// TwinCAT 3 PLC project Struckig
// Title: Struckig
// Company: Stefan Besler
// Author: Stefan Besler and contributers
// ProjectVersion: 0.15.5.0
// Description: Full port of pantor ruckig library (Community version) to IEC 61131-3 Structured Text. Online Trajectory Generation. Real-time. Time-optimal. Jerk-constrained.
// ProgramVersion: 3.1.4026.18
// project tree:
//   / Constants.TcGVL (not stored), ParameterList.TcGVL (not stored)
//   Struckig/Block/ BlockInterval.TcDUT (not stored), Block.TcDUT (not stored)
//   Struckig/BrakeProfile/ BrakeProfile.TcPOU (not stored)
//   Struckig/ Integrate.TcPOU (not stored), IOtg.TcIO (not stored), Otg1.TcPOU (not stored), Otg.TcPOU
//   Struckig/Math/ BubbleSortLreal.TcPOU (not stored), Ceil.TcPOU (not stored), Clamp.TcPOU (not stored), Fmod.TcPOU (not stored), IsNaN.TcPOU (not stored), IsInfinity.TcPOU (not stored), LrealBits.TcPOU (not stored), LrealFromBits.TcPOU (not stored), Power.TcPOU (not stored), Power2.TcPOU (not stored), Cbrt.TcPOU (not stored), Roots.TcPOU (not stored)
//   Struckig/Position/ PositionFirstOrderStep1.TcPOU (not stored), PositionFirstOrderStep2.TcPOU (not stored), PositionThirdOrderStep1.TcPOU (not stored), PositionSecondOrderStep1.TcPOU (not stored), PositionThirdOrderStep2.TcPOU (not stored), PositionSecondOrderStep2.TcPOU (not stored)
//   Struckig/Profile/ ProfileDesc.TcPOU (not stored)
//   Struckig/Profile/_DataTypes/ ProfileBound.TcDUT (not stored), ProfileDirection.TcDUT (not stored), ProfileControlSigns.TcDUT (not stored), ReachedLimits.TcDUT (not stored)
//   Struckig/Velocity/ VelocitySecondOrderStep2.TcPOU (not stored), VelocityThirdOrderStep1.TcPOU (not stored), VelocitySecondOrderStep1.TcPOU (not stored), VelocityThirdOrderStep2.TcPOU (not stored)
//   Struckig/_DataTypes/ ControlInterfaceType.TcDUT (not stored), DiscretizationType.TcDUT (not stored), SynchronizationType.TcDUT (not stored), TrajectoryErrorCode.TcDUT (not stored), TrajectoryState.TcDUT (not stored)

// ---- Struckig/Otg.TcPOU
// Struckig
// Copyright (C) 2022 Stefan Besler

// This program is free software: you can redistribute it and/or modify
// it under the terms of the GNU General Public License as published by
// the Free Software Foundation, either version 3 of the License, or
// (at your option) any later version.

// This program is distributed in the hope that it will be useful,
// but WITHOUT ANY WARRANTY; without even the implied warranty of
// MERCHANTABILITY or FITNESS FOR A PARTICULAR PURPOSE.  See the
// GNU General Public License for more details.
//
// You should have received a copy of the GNU General Public License
// along with THIS PROGRAM.  IF NOT, see <http://www.gnu.org/licenses/>.
{attribute 'conditionalshow_all_locals'}
FUNCTION_BLOCK Otg IMPLEMENTS IOtg
VAR_INPUT
  CycleTime : LREAL;
  Dofs : INT;
  Enabled : ARRAY[0..ParameterList.MaxDoFs] OF BOOL;  
  ControlInterface : ControlInterfaceType := ControlInterfaceType.Position; //< The default position interface controls the full kinematic state.
  Synchronization : SynchronizationType := SynchronizationType.TimeSync; //< Synchronization behavior of multiple DoFs
  PerDofControlInterface : ARRAY[0..ParameterList.MaxDoFs] OF ControlInterfaceType; //< Per-DoF control interface (overwrites global ControlInterface)
  PerDofSynchronization: ARRAY[0..ParameterList.MaxDoFs] OF SynchronizationType; //< Per-DoF synchronization (overwrites global Synchronization)
  Discretization : DiscretizationType; //< Whether the duration should be a discrete multiple of the control cycle (off by default)
  CurrentPosition, CurrentVelocity, CurrentAcceleration : ARRAY[0..ParameterList.MaxDoFs] OF LREAL; //< Current state
  TargetPosition, TargetVelocity, TargetAcceleration : ARRAY[0..ParameterList.MaxDoFs] OF LREAL; //< Target state
  MaxVelocity : ARRAY[0..ParameterList.MaxDoFs] OF LREAL; //< Kinematic constraints
  MaxAcceleration : ARRAY[0..ParameterList.MaxDoFs] OF LREAL; //< Kinematic constraints, defaults to Infinity (Struckig.Constants.Infinity)
  MaxJerk : ARRAY[0..ParameterList.MaxDoFs] OF LREAL; //< Kinematic constraints, defaults to Infinity (Struckig.Constants.Infinity)
  MinVelocity, MinAcceleration : ARRAY[0..ParameterList.MaxDoFs] OF LREAL; //< Optional kindematic constraints
  MinDuration : LREAL := 0; //< Optional minimum duration of a trajectory. This is only considered if the Synchronization type is not none
  EnableAutoPropagate : BOOL; //< If set to true, PassOutputToInput is automatically called internally after calling the function block's body
END_VAR
VAR_OUTPUT
  NewPosition, NewVelocity, NewAcceleration, NewJerk : ARRAY[0..ParameterList.MaxDoFs] OF LREAL;
  NewCalculation : BOOL; //< Was a new trajectory calculation performed in the last cycle?
  CurrentTime : LREAL;
END_VAR
VAR
  _duration : LREAL;
  _state : TrajectoryState;  
  _inputInitialized : BOOL := FALSE;
  _newSection : INT; //< not used in Struckig, ruckig pro feature
  _blocks : ARRAY[0..ParameterList.MaxDoFs] OF Block;  
  _profiles : ARRAY[0..ParameterList.MaxDoFs] OF ProfileDesc;
  _independentMinDurations : ARRAY[0..ParameterList.MaxDoFs] OF LREAL;
  
  _positionThirdOrderStep1 : PositionThirdOrderStep1;
  _positionThirdOrderStep2 : PositionThirdOrderStep2;
  _velocityThirdOrderStep1 : VelocityThirdOrderStep1;
  _velocityThirdOrderStep2 : VelocityThirdOrderStep2;
  
  _positionSecondOrderStep1 : PositionSecondOrderStep1;
  _positionSecondOrderStep2 : PositionSecondOrderStep2;
  _velocitySecondOrderStep1 : VelocitySecondOrderStep1;
  _velocitySecondOrderStep2 : VelocitySecondOrderStep2;
  
  _positionFirstOrderStep1 : PositionFirstOrderStep1;
  _positionFirstOrderStep2 : PositionFirstOrderStep2;  
  
  _inp_min_velocity, _inp_min_acceleration : ARRAY[0..ParameterList.MaxDoFs] OF LREAL;
  _inp_per_dof_control_interface : ARRAY[0..ParameterList.MaxDoFs] OF ControlInterfaceType; //< Per-DoF control interface
  _inp_per_dof_synchronization : ARRAY[0..ParameterList.MaxDoFs] OF SynchronizationType; //< Per-DoF synchronization
  
  _dofs, _dofsEnd : INT;
  _enabled : ARRAY[0..ParameterList.MaxDoFs] OF BOOL;  
  _controlInterface : ControlInterfaceType := ControlInterfaceType.Position; //< The default position interface controls the full kinematic state.
  _synchronization : SynchronizationType := SynchronizationType.TimeSync; //< Synchronization behavior of multiple DoFs
  _perDofControlInterface : ARRAY[0..ParameterList.MaxDoFs] OF ControlInterfaceType; //< Per-DoF control interface
  _perDofSynchronization: ARRAY[0..ParameterList.MaxDoFs] OF SynchronizationType; //< Per-DoF synchronization
  _discretization : DiscretizationType; //< Whether the duration should be a discrete multiple of the control cycle (off by default)
  _currentPosition, _currentVelocity, _currentAcceleration : ARRAY[0..ParameterList.MaxDoFs] OF LREAL; //< Current state
  _targetPosition, _targetVelocity, _targetAcceleration : ARRAY[0..ParameterList.MaxDoFs] OF LREAL; //< Target state
  _maxVelocity, _maxAcceleration, _maxJerk : ARRAY[0..ParameterList.MaxDoFs] OF LREAL; //< Kinematic constraints
  _new_phase_control : ARRAY[0..ParameterList.MaxDoFs] OF LREAL;
  _minVelocity, _minAcceleration : ARRAY[0..ParameterList.MaxDoFs] OF LREAL; //< Optional kindematic constraints
  _minDuration : LREAL := 0; //< Optional minimum duration of a trajectory. This is only considered if the Synchronization type is not none
  _dt : LREAL; //< Time step between updates (cycle time) in [s]
  _errorId : INT;
  _errorMessage : STRING(255);
END_VAR

NewCalculation := FALSE;
SetBusy(TRUE);

IF NOT _inputInitialized OR_ELSE HasChanged() 
THEN
  _dofsEnd := Dofs - 1; // for looping

  Calculate();
  IF State = TrajectoryState.Error THEN
    RETURN;
  END_IF

  // Store the desired state to check for potential changes
  _dofs := Dofs;
  _enabled := Enabled;
  _controlInterface := ControlInterface;
  _synchronization := Synchronization;
  _discretization := Discretization;
  _currentPosition := CurrentPosition;
  _currentVelocity := CurrentVelocity;
  _currentAcceleration := CurrentAcceleration;
  _targetPosition := TargetPosition;
  _targetVelocity := TargetVelocity;
  _targetAcceleration := TargetAcceleration;
  _maxVelocity := MaxVelocity;
  _maxAcceleration := MaxAcceleration;
  _maxJerk := MaxJerk;
  _minVelocity := MinVelocity;
  _minAcceleration := MinAcceleration;
  _minDuration := MinDuration;
  _perDofControlInterface := PerDofControlInterface;
  _perDofSynchronization := PerDofSynchronization;
  _dt := CycleTime;
  _inputInitialized := TRUE;
  CurrentTime := 0.0;
  NewCalculation := TRUE;  
END_IF

CurrentTime := CurrentTime + _dt;
AtTime(CurrentTime, ADR(NewPosition), ADR(NewVelocity), ADR(NewAcceleration), ADR(NewJerk), ADR(_newSection));

_currentPosition := NewPosition;
_currentVelocity := NewVelocity;
_currentAcceleration := NewAcceleration;

IF CurrentTime > _duration THEN
  _state := TrajectoryState.Idle;
END_IF

IF EnableAutoPropagate
THEN
  PassOutputToInput();
END_IF

METHOD PROTECTED AbortErrorId
VAR_INPUT
  errorId : INT;
END_VAR
VAR_IN_OUT CONSTANT  
  message : STRING;
END_VAR
_state := TrajectoryState.Error;
_errorMessage := message;
_errorId := errorId;
END_METHOD

/// Get the kinematic state at a given time
{attribute 'conditionalshow'}
METHOD AtTime
VAR_INPUT
  t : LREAL;
  new_position : POINTER TO LREAL;
  new_velocity : POINTER TO LREAL;
  new_acceleration : POINTER TO LREAL;
  new_jerk : POINTER TO LREAL;
  new_section : POINTER TO INT;
END_VAR
VAR
  dof : INT;
  p : REFERENCE TO ProfileDesc;
  t_diff : LREAL;
  index : INT;
END_VAR
IF (t >= Duration) THEN
  // Keep constant acceleration
  //new_section := 1;
  FOR dof:=0 TO _dofsEnd DO
    Integrate(t - (_profiles[dof].Brake.Duration + _profiles[dof].t_sum[6]), _profiles[dof].p[7], _profiles[dof].v[7], _profiles[dof].a[7], 0, p:=new_position[dof], v:=new_velocity[dof], a:=new_acceleration[dof]);
    new_jerk[dof] := 0;
  END_FOR
  RETURN;
END_IF

//new_section := 0;
FOR dof:=0 TO _dofsEnd DO
  p REF= _profiles[dof];

  t_diff := t;
  
  // Brake pre-trajectory
  IF (p.Brake.Duration > 0) THEN
    IF (t_diff < p.Brake.Duration) THEN
      index := SEL(t_diff < p.Brake.t[0], 1, 0);
      IF (index > 0) THEN
        t_diff := t_diff - p.Brake.t[index - 1];
      END_IF

      Integrate(t_diff, p.Brake.p[index], p.Brake.v[index], p.Brake.a[index], p.Brake.j[index], p:=new_position[dof], v:=new_velocity[dof], a:=new_acceleration[dof]);
      new_jerk[dof] := p.Brake.j[index];
      CONTINUE;
    ELSE
      t_diff := t_diff - p.Brake.Duration;
    END_IF
  END_IF
  
// Accel post-trajectory
// if (new_section == profiles.size() - 1 && p.accel.duration > 0) {
//     if (t_diff_dof > p.t_sum[6]) {
//         const size_t index = (t_diff_dof < p.accel.t[0]) ? 1 : 0;
//         if (index > 0) {
//             t_diff_dof -= p.accel.t[index - 1];
//         }

//         std::tie(new_position[dof], new_velocity[dof], new_acceleration[dof]) = integrate(t_diff_dof, p.accel.p[index], p.accel.v[index], p.accel.a[index], p.accel.j[index]);
//         continue;
//     }
// }

  // Non-time synchronization
  IF (t_diff >= p.t_sum[6]) THEN
    // Keep constant acceleration
    Integrate(t_diff - p.t_sum[6], p.p[7], p.v[7], p.a[7], 0, p:=new_position[dof], v:=new_velocity[dof], a:=new_acceleration[dof]);
    new_jerk[dof] := 0;    
    CONTINUE;
  END_IF

  FOR index:=0 TO 6 DO
    IF p.t_sum[index] > t_diff
    THEN
      EXIT;
    END_IF
	END_FOR
  
  IF (index > 0) THEN
    t_diff := t_diff - p.t_sum[index - 1];
  END_IF

  Integrate(t_diff, p.p[index], p.v[index], p.a[index], p.j[index], p:=new_position[dof], v:=new_velocity[dof], a:=new_acceleration[dof]);
  new_jerk[dof] := p.j[index];      
END_FOR
END_METHOD

/// Get the kinematic state and current section at a given time without vectors for a single DoF.
/// Using this method is only allowed for DoF = 1, for higher degrees of freedom use
/// [AtTime](xref:Struckig.Otg#AtTime). Using this method for DoF > 0 will not yield any result
{attribute 'conditionalshow'}
METHOD AtTime1
VAR_INPUT
  t : LREAL;
  new_position : REFERENCE TO LREAL;
  new_velocity : REFERENCE TO LREAL;
  new_acceleration : REFERENCE TO LREAL;
  new_jerk : REFERENCE TO LREAL;  
END_VAR
IF _dofs = 1
THEN
  AtTime(t, ADR(new_position), ADR(new_velocity), ADR(new_acceleration), ADR(new_jerk), 0);
END_IF
END_METHOD

METHOD PRIVATE Calculate
VAR_INST
  dof, i : INT;
  p, p_limiting : REFERENCE TO ProfileDesc;
  found_profile : BOOL;
  limiting_dof : INT := -1; // The DoF that doesn't need step 2
  discrete_duration, found_synchronization, found_time_synchronization : BOOL;
  t_profile : LREAL;
  noneSynchronizationCount, phaseSychronizations, phaseOrNoneSychronizationCount : INT;
  has_zero_limits : BOOL;
END_VAR
SetBusy(TRUE);
IF NOT ValidateInputOrAbort(checkCurrentStateWithinLimits:=FALSE, checkTargetStateWithinLimits:=TRUE)
THEN
  RETURN;
END_IF

FOR dof:=0 TO _dofsEnd
DO
  p REF=_profiles[dof];
  
  _inp_min_velocity[dof] := SEL(ABS(MinVelocity[dof]) < Constants.Epsilon, MinVelocity[dof], -MaxVelocity[dof]);
  _inp_min_acceleration[dof] := SEL(ABS(MinAcceleration[dof]) < Constants.Epsilon, MinAcceleration[dof], -MaxAcceleration[dof]);
  _inp_per_dof_control_interface[dof] := SEL(PerDofControlInterface[dof] = ControlInterfaceType.Undefined, PerDofControlInterface[dof], ControlInterface);
  _inp_per_dof_synchronization[dof] := SEL(PerDofSynchronization[dof] = SynchronizationType.Undefined, PerDofSynchronization[dof], Synchronization); 
  
  IF NOT Enabled[dof]
  THEN
    p.p[7] := CurrentPosition[dof];
    p.v[7] := CurrentVelocity[dof];
    p.a[7] := CurrentAcceleration[dof];    
    p.t_sum[6] := 0.0;
    _blocks[dof].Tmin := 0.0;
    _blocks[dof].A.IsUsed := FALSE;
    _blocks[dof].B.IsUsed := FALSE;    
    CONTINUE;
	END_IF
  
  CASE _inp_per_dof_control_interface[dof]
  OF
    ControlInterfaceType.Position:
    
      IF NOT IsInfinity(MaxJerk[dof])
      THEN
        p.Brake.PositionBrakeTrajectory(CurrentVelocity[dof], CurrentAcceleration[dof], MaxVelocity[dof], _inp_min_velocity[dof], MaxAcceleration[dof], _inp_min_acceleration[dof], MaxJerk[dof]);
      ELSIF NOT IsInfinity(MaxAcceleration[dof])
      THEN
        p.Brake.SecondOrderPositionBrakeTrajectory(CurrentVelocity[dof], MaxVelocity[dof], _inp_min_velocity[dof], MaxAcceleration[dof], _inp_min_acceleration[dof]);
      END_IF    

      p.SetBoundaryPosition(CurrentPosition[dof], CurrentVelocity[dof], CurrentAcceleration[dof], TargetPosition[dof], TargetVelocity[dof], TargetAcceleration[dof]);

    ControlInterfaceType.Velocity:
      IF NOT IsInfinity(MaxJerk[dof])
      THEN    
        p.Brake.VelocityBrakeTrajectory(CurrentVelocity[dof], CurrentAcceleration[dof], MaxAcceleration[dof], _inp_min_acceleration[dof], MaxJerk[dof]);
      ELSIF NOT IsInfinity(MaxAcceleration[dof])
      THEN
        p.Brake.SecondOrderVelocityBrakeTrajectory();        
      END_IF
      
      p.SetBoundaryVelocity(CurrentPosition[dof], CurrentVelocity[dof], CurrentAcceleration[dof], TargetVelocity[dof], TargetAcceleration[dof]);      
	END_CASE
  
  IF NOT IsInfinity(MaxJerk[dof])
  THEN
    p.Brake.Finalize(p.p[0], p.v[0], p.a[0]);
  ELSIF NOT IsInfinity(MaxAcceleration[dof])
  THEN
    p.Brake.FinalizeSecondOrder(p.p[0], p.v[0], p.a[0]);    
  END_IF

  CASE _inp_per_dof_control_interface[dof]
  OF
    ControlInterfaceType.Position:
      IF NOT IsInfinity(MaxJerk[dof])
      THEN
        _positionThirdOrderStep1.Set(p.p[0], p.v[0], p.a[0], p.pf, p.vf, p.af, MaxVelocity[dof], _inp_min_velocity[dof], MaxAcceleration[dof], _inp_min_acceleration[dof], MaxJerk[dof]);
        found_profile := _positionThirdOrderStep1.Get(p, _blocks[dof]);      
      ELSIF NOT IsInfinity(MaxAcceleration[dof])
      THEN
        _positionSecondOrderStep1.Set(p.p[0], p.v[0], p.pf, p.vf, MaxVelocity[dof], _inp_min_velocity[dof], MaxAcceleration[dof], _inp_min_acceleration[dof]);
        found_profile := _positionSecondOrderStep1.Get(p, _blocks[dof]);          
      ELSE
        _positionFirstOrderStep1.Set(p.p[0], p.pf, MaxVelocity[dof], _inp_min_velocity[dof]);
        found_profile := _positionFirstOrderStep1.Get(p, _blocks[dof]);          
      END_IF

    ControlInterfaceType.Velocity:
      IF NOT IsInfinity(MaxJerk[dof])
      THEN    
        _velocityThirdOrderStep1.Set(p.v[0], p.a[0], p.vf, p.af, MaxAcceleration[dof], _inp_min_acceleration[dof], MaxJerk[dof]);
        found_profile := _velocityThirdOrderStep1.Get(p, _blocks[dof]);
      ELSIF NOT IsInfinity(MaxAcceleration[dof])
      THEN
        _velocitySecondOrderStep1.Set(p.v[0], p.vf, MaxAcceleration[dof], _inp_min_acceleration[dof]);
        found_profile := _velocitySecondOrderStep1.Get(p, _blocks[dof]);    
      END_IF  
	END_CASE
  
  IF NOT found_profile
  THEN
    has_zero_limits := (MaxAcceleration[dof] = 0.0 OR_ELSE _inp_min_acceleration[dof] = 0.0 OR_ELSE MaxJerk[dof] = 0.0);
    IF has_zero_limits
    THEN
      AbortErrorId(TrajectoryErrorCode.ZeroLimitsConflict, '');
      RETURN;
    ELSE 
      AbortErrorId(TrajectoryErrorCode.CalculateStep1Failed, '');      
      RETURN;
    END_IF
	END_IF

  _independentMinDurations[dof] := _blocks[dof].Tmin;
END_FOR


discrete_duration := (Discretization = DiscretizationType.Discrete);

IF (dofs = 0 AND_THEN MinDuration <> 0 AND_THEN discrete_duration <> 0)
THEN 
  _duration := _blocks[0].Tmin;
  _profiles[0] := _blocks[0].Pmin;
  RETURN;
END_IF

found_synchronization := Synchronize(discrete_duration, MinDuration, _duration, limiting_dof);
IF NOT found_synchronization
THEN
  has_zero_limits := FALSE;
  FOR i:=0 TO _dofsEnd
  DO
    IF MaxAcceleration[dof] = 0.0 OR_ELSE _inp_min_acceleration[dof] = 0.0 OR_ELSE MaxJerk[dof] = 0.0
    THEN
      has_zero_limits := TRUE;
      EXIT;
    END_IF
  END_FOR
      
  IF has_zero_limits
  THEN
    AbortErrorId(TrajectoryErrorCode.ZeroLimitsConflictInSynchronization, '');
    RETURN;
  ELSE
    AbortErrorId(TrajectoryErrorCode.SynchronizationFailed, '');
    RETURN;    
	END_IF    
END_IF

// None Synchronization
FOR dof:=0 TO _dofsEnd
DO
  IF Enabled[dof] AND_THEN _inp_per_dof_synchronization[dof] = SynchronizationType.None
  THEN
    _profiles[dof] := _blocks[dof].Pmin;
    IF _blocks[dof].Tmin > Duration
    THEN
      _duration := _blocks[dof].Tmin;
      limiting_dof := dof;
    END_IF
  END_IF
END_FOR

IF (Duration = 0.0) THEN
  // Copy all profiles for end state
  FOR dof:=0 TO _dofsEnd
  DO
    _profiles[dof] := _blocks[dof].Pmin;
  END_FOR
  RETURN;
END_IF

noneSynchronizationCount := -1;
phaseSychronizations := -1;
phaseOrNoneSychronizationCount := -1;
FOR dof:=0 TO _dofsEnd DO 
  IF _inp_per_dof_synchronization[dof] = SynchronizationType.None
  THEN
    noneSynchronizationCount := noneSynchronizationCount + 1;
    phaseOrNoneSychronizationCount := phaseOrNoneSychronizationCount + 1;
  ELSIF _inp_per_dof_synchronization[dof] = SynchronizationType.Phase
  THEN
    phaseOrNoneSychronizationCount := phaseOrNoneSychronizationCount + 1;
    phaseSychronizations := phaseSychronizations + 1;
  END_IF
END_FOR

IF NOT discrete_duration AND_THEN noneSynchronizationCount = _dofsEnd
THEN
  RETURN;
END_IF

IF limiting_dof >= 0 AND_THEN phaseSychronizations >= 0 THEN
  p_limiting REF= _profiles[limiting_dof];
  IF IsInputCollinear(p_limiting.Direction, limiting_dof, _new_phase_control) THEN
    found_time_synchronization := TRUE;
    FOR dof:=0 TO _dofsEnd DO
      IF NOT Enabled[dof] OR_ELSE dof = limiting_dof OR_ELSE _inp_per_dof_synchronization[dof] <> SynchronizationType.Phase THEN
        CONTINUE;
      END_IF

      p REF= _profiles[dof];
      t_profile := Duration - p.Brake.Duration - p.Accel.Duration;

      p.t := p_limiting.t; // Copy timing information from limiting DoF
      p.ControlSigns := p_limiting.ControlSigns;

      CASE _inp_per_dof_control_interface[dof]
      OF
        ControlInterfaceType.Position:
          CASE p.ControlSigns
          OF
            ProfileControlSigns.Uddu:
            
              IF NOT IsInfinity(MaxJerk[dof])
              THEN
                IF NOT p.CheckWithTiming2(ProfileControlSigns.Uddu, ReachedLimits.None, t_profile, _new_phase_control[dof], MaxVelocity[dof], _inp_min_velocity[dof], MaxAcceleration[dof], _inp_min_acceleration[dof], MaxJerk[dof])
                THEN
                  found_time_synchronization := FALSE;                        
                END_IF
              ELSIF NOT IsInfinity(MaxAcceleration[dof])
              THEN
                IF NOT p.CheckForSecondOrderWithTiming2(ProfileControlSigns.Uddu, ReachedLimits.None, t_profile, _new_phase_control[dof], -_new_phase_control[dof], MaxVelocity[dof], _inp_min_velocity[dof], MaxAcceleration[dof], _inp_min_acceleration[dof])
                THEN
                  found_time_synchronization := FALSE;                        
                END_IF
              ELSE
                IF NOT p.CheckForFirstOrderWithTiming2(ProfileControlSigns.Uddu, ReachedLimits.None, t_profile, _new_phase_control[dof], MaxVelocity[dof], _inp_min_velocity[dof])
                THEN
                  found_time_synchronization := FALSE;                        
                END_IF
              END_IF
            
            ProfileControlSigns.Udud:
              IF NOT IsInfinity(MaxJerk[dof])
              THEN            
                IF NOT p.CheckWithTiming2(ProfileControlSigns.Udud, ReachedLimits.None, t_profile, _new_phase_control[dof], MaxVelocity[dof], _inp_min_velocity[dof], MaxAcceleration[dof], _inp_min_acceleration[dof], MaxJerk[dof])
                THEN            
                  found_time_synchronization := FALSE;
                END_IF
              ELSE
                IF NOT p.CheckForSecondOrderWithTiming2(ProfileControlSigns.Udud, ReachedLimits.None, t_profile, _new_phase_control[dof], -_new_phase_control[dof], MaxVelocity[dof], _inp_min_velocity[dof], MaxAcceleration[dof], _inp_min_acceleration[dof])
                THEN
                  found_time_synchronization := FALSE;                        
                END_IF
              END_IF                
          END_CASE
        
        ControlInterfaceType.Velocity:
          CASE p.ControlSigns
          OF
            ProfileControlSigns.Uddu:
            
              IF NOT IsInfinity(MaxJerk[dof])
              THEN  
                IF NOT p.CheckForVelocityWithTiming(ProfileControlSigns.Uddu, ReachedLimits.None, _new_phase_control[dof], MaxAcceleration[dof], _inp_min_acceleration[dof], MaxJerk[dof])
                THEN
                  found_time_synchronization := FALSE;                        
                END_IF
              ELSE
                IF NOT p.CheckForSecondOrderVelocityWithTiming2(ProfileControlSigns.Uddu, ReachedLimits.None, t_profile, _new_phase_control[dof], MaxAcceleration[dof], _inp_min_acceleration[dof])
                THEN
                  found_time_synchronization := FALSE;                        
                END_IF
              END_IF
          
            ProfileControlSigns.Udud:
            
              IF NOT IsInfinity(MaxJerk[dof])
              THEN             
                IF NOT p.CheckForVelocityWithTiming(ProfileControlSigns.Udud, ReachedLimits.None, _new_phase_control[dof], MaxAcceleration[dof], _inp_min_acceleration[dof], MaxJerk[dof])
                THEN            
                  found_time_synchronization := FALSE;
                END_IF
              ELSE
                IF NOT p.CheckForSecondOrderVelocityWithTiming2(ProfileControlSigns.Udud, ReachedLimits.None, t_profile, _new_phase_control[dof], MaxAcceleration[dof], _inp_min_acceleration[dof])
                THEN
                  found_time_synchronization := FALSE;                        
                END_IF
              END_IF                
          END_CASE        
      END_CASE
  

      p.Limits := p_limiting.Limits; // After check method call to set correct limits
    END_FOR

    IF found_time_synchronization AND_THEN phaseOrNoneSychronizationCount = _dofsEnd  THEN
      RETURN;
    END_IF
  END_IF
END_IF

// Time Synchronization
FOR dof:=0 TO _dofsEnd
DO
  IF NOT Enabled[dof] OR_ELSE ((dof = limiting_dof OR_ELSE _inp_per_dof_synchronization[dof] = SynchronizationType.None) AND_THEN NOT discrete_duration) THEN
    CONTINUE;
  END_IF
  
  p REF= _profiles[dof];
  t_profile := Duration - p.Brake.Duration - p.Accel.Duration;
  
  IF (_inp_per_dof_synchronization[dof] = SynchronizationType.TimeIfNecessarySync AND_THEN ABS(TargetVelocity[dof]) < Constants.Epsilon AND_THEN ABS(CurrentAcceleration[dof]) < Constants.Epsilon) THEN
      p := _blocks[dof].Pmin;
      CONTINUE;
  END_IF
  
  // Check if the final time corresponds to an extremal profile calculated in step 1
  // Use 2*eps because of numerical robustness in duration discretization
  IF (ABS(t_profile - _blocks[dof].Tmin) < Constants.Epsilon) THEN
      p := _blocks[dof].Pmin;
      CONTINUE;
  ELSIF (_blocks[dof].A.IsUsed AND_THEN ABS(t_profile - _blocks[dof].A.Right) < 2 * Constants.Epsilon16)
  THEN
      p := _blocks[dof].A.Profile;
      CONTINUE;
  ELSIF (_blocks[dof].B.IsUsed AND_THEN ABS(t_profile - _blocks[dof].B.Right) < 2 * Constants.Epsilon16)
  THEN
      p := _blocks[dof].B.Profile;
      CONTINUE;
  END_IF
  
  CASE (_inp_per_dof_control_interface[dof])
  OF  
    ControlInterfaceType.Position: 
    
      IF NOT IsInfinity(MaxJerk[dof])
      THEN       
        _positionThirdOrderStep2.Set(t_profile, p.p[0], p.v[0], p.a[0], p.pf, p.vf, p.af, MaxVelocity[dof], _inp_min_velocity[dof], MaxAcceleration[dof], _inp_min_acceleration[dof], MaxJerk[dof]);
        found_time_synchronization := _positionThirdOrderStep2.Get(p);
      ELSIF NOT IsInfinity(MaxAcceleration[dof])
      THEN
        _positionSecondOrderStep2.Set(t_profile, p.p[0], p.v[0], p.pf, p.vf, MaxVelocity[dof], _inp_min_velocity[dof], MaxAcceleration[dof], _inp_min_acceleration[dof]);
        found_time_synchronization := _positionSecondOrderStep2.Get(p);        
      ELSE
        _positionFirstOrderStep2.Set(t_profile, p.p[0], p.pf, MaxVelocity[dof], _inp_min_velocity[dof]);
        found_time_synchronization := _positionFirstOrderStep2.Get(p);        
      END_IF

    ControlInterfaceType.Velocity: 
      IF NOT IsInfinity(MaxJerk[dof])
      THEN    
        _velocityThirdOrderStep2.Set(t_profile, p.v[0], p.a[0], p.vf, p.af, MaxAcceleration[dof], _inp_min_acceleration[dof], MaxJerk[dof]);
        found_time_synchronization := _velocityThirdOrderStep2.Get(p);
      ELSE
        _velocitySecondOrderStep2.Set(t_profile, p.v[0], p.vf, MaxAcceleration[dof], _inp_min_acceleration[dof]);
        found_time_synchronization := _velocitySecondOrderStep2.Get(p);
      END_IF
  END_CASE

  IF NOT found_time_synchronization
  THEN
    AbortErrorId(TrajectoryErrorCode.SynchronizationFailed, '');
    RETURN;
  END_IF
END_FOR
END_METHOD

/// This method simply calls the body of the function block
METHOD Cyclic
VAR_INPUT
END_VAR
THIS^();
END_METHOD

PROPERTY Duration : LREAL
GET
Duration := _duration;
END_GET
END_PROPERTY

METHOD ErrorCode : TrajectoryErrorCode
VAR_INPUT
END_VAR
ErrorCode := _errorId;
END_METHOD

METHOD ErrorMessage : STRING(255)
VAR_INPUT
END_VAR
IF _errorMessage = ''
THEN
  CASE _errorId
  OF
    TrajectoryErrorCode.CalculateStep1Failed: ErrorMessage := 'Trajectory generation failed in step1';
    TrajectoryErrorCode.InvalidInput: ErrorMessage := 'Trajectory-generation invalid input';
    TrajectoryErrorCode.SynchronizationFailed: ErrorMessage := 'Trajectory-generation synchronization failed';
    TrajectoryErrorCode.ZeroLimitsConflict: ErrorMessage := 'Zero limits conflict in step 1';
    TrajectoryErrorCode.ZeroLimitsConflictInSynchronization: ErrorMessage := 'Zero limits conflict with other degrees of freedom in time synchronization';

  ELSE
    IF State = TrajectoryState.Error
    THEN
      ErrorMessage := 'Unknown error';
    END_IF
  END_CASE
ELSE
  ErrorMessage := _errorMessage;
END_IF
END_METHOD

METHOD FB_init : BOOL
VAR_INPUT
	bInitRetains : BOOL; // if TRUE, the retain variables are initialized (warm start / cold start)
	bInCopyCode : BOOL;  // if TRUE, the instance afterwards gets moved into the copy code (online change)
  cycletime : LREAL;
  dofs : SINT;
END_VAR
VAR
  i : INT;
  blockSize : UDINT := SIZEOF(Block)*SINT_TO_UDINT(dofs);
  profileSize : UDINT :=  SIZEOF(ProfileDesc)*SINT_TO_UDINT(dofs);  
END_VAR
THIS^.Dofs := dofs;

FOR i:=0 TO ParameterList.MaxDoFs
DO
  Enabled[i] := i < dofs;
  MaxAcceleration[i] := Constants.Infinity;  
  MaxJerk[i] := Constants.Infinity;
END_FOR
_dt := THIS^.CycleTime := cycletime;
END_METHOD

METHOD PRIVATE HasChanged : BOOL
VAR
  i : INT;  
END_VAR
IF _dofs <> Dofs
THEN
  HasChanged := TRUE;
  RETURN;
END_IF

FOR i:=0 TO _dofsEnd
DO
  IF NOT (_currentPosition[i] = CurrentPosition[i] AND_THEN
     _currentVelocity[i] = CurrentVelocity[i] AND_THEN
     _currentAcceleration[i] = CurrentAcceleration[i] AND_THEN
     _targetPosition[i] = TargetPosition[i] AND_THEN
     _targetVelocity[i] = TargetVelocity[i] AND_THEN
     _targetAcceleration[i] = TargetAcceleration[i] AND_THEN
     _maxVelocity[i] = MaxVelocity[i] AND_THEN
     _maxAcceleration[i] = MaxAcceleration[i] AND_THEN
     _maxJerk[i] = MaxJerk[i] AND_THEN
     _enabled[i] = Enabled[i] AND_THEN
     _minVelocity[i] = MinVelocity[i] AND_THEN
     _minAcceleration[i] = MinAcceleration[i] AND_THEN
     _perDofControlInterface[i] = PerDofControlInterface[i] AND_THEN
     _perDofSynchronization[i] = PerDofSynchronization[i])
  THEN
    HasChanged := TRUE;  
    RETURN;
	END_IF
END_FOR

IF NOT (_controlInterface = ControlInterface AND_THEN
   _synchronization = Synchronization AND_THEN
   _discretization = Discretization AND_THEN
   _minDuration = MinDuration)   
THEN
  HasChanged := TRUE;
  RETURN;
END_IF
END_METHOD

METHOD INTERNAL IsBlocked : BOOL
VAR_INPUT
  block : REFERENCE TO Block;
  t : LREAL;
END_VAR
IsBlocked := (t < block.Tmin) OR_ELSE (block.A.IsUsed AND_THEN block.A.Left < t AND_THEN t < block.A.Right) OR_ELSE (block.B.IsUsed AND_THEN block.B.Left < t AND_THEN t < block.B.Right);
END_METHOD

/// Is the trajectory (in principle) phase synchronizable?
METHOD INTERNAL IsInputCollinear : BOOL
VAR_INPUT
  limitingDirection : ProfileDirection;
  limitingDof : INT;
  new_phase_control : REFERENCE TO ARRAY[0..ParameterList.MaxDoFs] OF LREAL;
END_VAR
VAR_INST
  scale_dof : INT := -1;
  dof : INT;
  pd : ARRAY[0..ParameterList.MaxDoFs] OF LREAL;
  scale_vector : POINTER TO LREAL;
  pd_scale, v0_scale, a0_scale, vf_scale, af_scale, scale, scale_limiting, current_scale : LREAL;
  control_limiting : LREAL;
END_VAR
// Check that vectors pd, v0, a0, vf, af are collinear
FOR dof:=0 TO _dofsEnd
DO
  pd[dof] := TargetPosition[dof] - CurrentPosition[dof];
END_FOR

scale_dof := -1;
FOR dof:=0 TO _dofsEnd
DO
  IF _inp_per_dof_synchronization[dof] <> SynchronizationType.Phase
  THEN
    CONTINUE;
	END_IF
  
  IF _inp_per_dof_control_interface[dof] = ControlInterfaceType.Position AND_THEN ABS(pd[dof]) > Constants.Epsilon
  THEN
    scale_vector := ADR(pd);
    scale_dof := dof;
    EXIT;

  ELSIF ABS(CurrentVelocity[dof]) > Constants.Epsilon
  THEN
    scale_vector := ADR(CurrentVelocity);
    scale_dof := dof;
    EXIT;

  ELSIF ABS(CurrentAcceleration[dof]) >  Constants.Epsilon
  THEN
    scale_vector := ADR(CurrentAcceleration);
    scale_dof := dof;
    EXIT;
  
  ELSIF ABS(TargetVelocity[dof]) >  Constants.Epsilon
  THEN
    scale_vector := ADR(TargetVelocity);
    scale_dof := dof;
    EXIT;

  ELSIF ABS(TargetAcceleration[dof]) > Constants.Epsilon
  THEN
    scale_vector := ADR(TargetAcceleration);
    scale_dof := dof;
    EXIT;
  END_IF
END_FOR

IF scale_dof < 0
THEN
  RETURN; // Zero everywhere is in theory collinear, but that trivial case is better handled elsewhere
END_IF

scale := scale_vector[scale_dof];
pd_scale := pd[scale_dof] / scale;
v0_scale := CurrentVelocity[scale_dof] / scale;
vf_scale := TargetVelocity[scale_dof] / scale;
a0_scale := CurrentAcceleration[scale_dof] / scale;
af_scale := TargetAcceleration[scale_dof] / scale;

scale_limiting := scale_vector[limitingDof];
control_limiting := SEL(limitingDirection = ProfileDirection.Up, -MaxJerk[limitingDof], MaxJerk[limitingDof]);

IF IsInfinity(MaxJerk[limitingDof])
THEN
  control_limiting := SEL(limitingDirection = ProfileDirection.Up, _inp_min_acceleration[limitingDof], MaxAcceleration[limitingDof]);
END_IF

IF ABS(scale_limiting) < Constants.Epsilon
THEN
  RETURN;
END_IF

FOR dof:=0 TO _dofsEnd
DO
  IF _inp_per_dof_synchronization[dof] <> SynchronizationType.Phase
  THEN
    CONTINUE;
	END_IF
  
  current_scale := scale_vector[dof];
  IF (_inp_per_dof_control_interface[dof] = ControlInterfaceType.Position AND_THEN ABS(pd[dof] - pd_scale * current_scale) > Constants.Epsilon)
    OR_ELSE ABS(CurrentVelocity[dof] - v0_scale * current_scale) > Constants.Epsilon
    OR_ELSE ABS(CurrentAcceleration[dof] - a0_scale * current_scale) > Constants.Epsilon
    OR_ELSE ABS(TargetVelocity[dof] - vf_scale * current_scale) > Constants.Epsilon
    OR_ELSE ABS(TargetAcceleration[dof] - af_scale * current_scale) > Constants.Epsilon
  THEN
    RETURN;
	END_IF
  
  new_phase_control[dof] := control_limiting * current_scale / scale_limiting;
END_FOR

IsInputCollinear := TRUE;
END_METHOD

METHOD PassOutputToInput
VAR_INPUT
END_VAR
CurrentPosition := NewPosition;
CurrentVelocity := NewVelocity;
CurrentAcceleration := NewAcceleration;

// Remove first intermediate waypoint if section did change
// not supported in Struckig, this is a Ruckig Pro Feature
//IF HasSectionChanged AND_THEN IntermediatePositionCount > 0
//THEN
//  IntermediatePositionIndex := IntermediatePositionIndex + 1;
//END_IF
END_METHOD

/// Resets the instance (e.g. to force a new calculation on the next update).
/// This method can be used to trigger a new trajectory even if inputs do not change.
METHOD Reset
VAR_INPUT
END_VAR
_inputInitialized := FALSE;
END_METHOD

METHOD PROTECTED SetBusy
VAR_INPUT
  on : BOOL;
END_VAR
_state := TrajectoryState.Busy;
END_METHOD

PROPERTY State : TrajectoryState
GET
State := _state;
END_GET
END_PROPERTY

METHOD INTERNAL Synchronize : BOOL
VAR_INPUT
  discrete_duration : BOOL;
END_VAR
VAR_IN_OUT
  Tmin : LREAL;
  t_sync : LREAL;
  limiting_dof : INT;
END_VAR
VAR_INST
  possible_t_syncs : ARRAY [0..3*ParameterList.MaxDoFs] OF LREAL;
  idx : ARRAY [0..3*ParameterList.MaxDoFs] OF INT;  
  idx_end : INT;
  possible_t_sync : REFERENCE TO LREAL;
  any_interval : BOOL;
  dof : INT;
  i,j, h : INT;
  is_blocked : BOOL;
  remainder : LREAL;
END_VAR
// Possible t_syncs are the start times of the intervals and optional Tmin
any_interval := FALSE;
FOR dof := 0 TO _dofsEnd
DO
  // Ignore DoFs without synchronization here
  IF _inp_per_dof_synchronization[dof] = SynchronizationType.None
  THEN
    possible_t_syncs[dof] := 0;
    possible_t_syncs[Dofs + dof] := Constants.Infinity;
    possible_t_syncs[2 * Dofs + dof] := Constants.Infinity;
  ELSE
    possible_t_syncs[dof] := _blocks[dof].Tmin;
    possible_t_syncs[Dofs + dof] := SEL(_blocks[dof].A.IsUsed, Constants.Infinity, _blocks[dof].A.Right);
    possible_t_syncs[2 * Dofs + dof] := SEL(_blocks[dof].B.IsUsed, Constants.Infinity, _blocks[dof].B.Right);
    any_interval := any_interval OR_ELSE _blocks[dof].A.IsUsed OR_ELSE _blocks[dof].B.IsUsed;
  END_IF
END_FOR

possible_t_syncs[3 * Dofs] := SEL(Tmin = 0, Tmin, Constants.Infinity);
any_interval := any_interval OR_ELSE Tmin > 0;
IF discrete_duration
THEN
  FOR i:=0 TO 3*Dofs-1
  DO
    possible_t_sync REF= possible_t_syncs[i];
    IF possible_t_sync = Constants.Infinity
    THEN
      CONTINUE;
		END_IF
    
    remainder := Fmod(possible_t_sync, CycleTime); // in [0, delta_time)
    IF remainder > Constants.Epsilon16 THEN
      possible_t_sync := possible_t_sync + CycleTime - remainder;
    END_IF     
  END_FOR
END_IF

// Bubblesort possible_t_syncs from best to worst
idx_end := SEL(any_interval, _dofsEnd, 3*DOFs);
BubbleSortLreal(ADR(possible_t_syncs), idx_end, indicesSorted:=ADR(idx));

// Start at last tmin (or worse)
FOR i:=_dofsEnd TO idx_end
DO  
  possible_t_sync REF= possible_t_syncs[idx[i]];
  
  is_blocked := FALSE;
  FOR dof:=0 TO _dofsEnd
  DO
    IF _inp_per_dof_synchronization[dof] = SynchronizationType.None
    THEN
      CONTINUE;
		END_IF
    
    IF IsBlocked(_blocks[dof], possible_t_sync) 
    THEN
      is_blocked := TRUE;
      EXIT;
		END_IF
	END_FOR
  
  IF is_blocked OR_ELSE possible_t_sync < Tmin OR_ELSE possible_t_sync = Constants.Infinity
  THEN
    CONTINUE;
	END_IF
    
  t_sync := possible_t_sync;
  IF (idx[i] = 3*Dofs)  // Optional Tmin
  THEN
    limiting_dof := -1;
    Synchronize := TRUE;
    RETURN;
  END_IF

  limiting_dof := (idx[i] MOD Dofs);
  CASE TRUNC(idx[i] / Dofs)
  OF
    0: _profiles[limiting_dof] := _blocks[limiting_dof].Pmin;
    1: _profiles[limiting_dof] := _blocks[limiting_dof].A.Profile;
    2: _profiles[limiting_dof] := _blocks[limiting_dof].B.Profile;  
	END_CASE
  
  Synchronize := TRUE;
  RETURN;
  
END_FOR
END_METHOD

/// To check that *Struckig* is able to generate a trajectory before the actual calculation step,
/// ```st
/// ruckig.ValidateInput(input, currentState: FALSE, targetState: TRUE);
/// // returns boolean
/// ```
/// returns `FALSE` if an input is not valid. The two boolean arguments check that the current or target state are 
/// within the limits. The check includes a typical catch of jerk-limited trajectory generation: 
/// When the current state is at maximal velocity, any positive acceleration will inevitable lead to a velocity violation 
/// *at a future timestep*. In general, this condition is fulfilled when
/// ```
/// Abs(acceleration) <= Sqrt(2 * max_jerk * (max_velocity - Abs(velocity))).
/// ```
/// If both arguments are set to true, the calculated trajectory is guaranteed to be *within the kinematic limits throughout* 
/// its duration. Also, note that there are range constraints of the input due to numerical reasons, see below for more details.
{attribute 'conditionalshow'}
METHOD ValidateInput : BOOL
VAR_INPUT
  checkCurrentStateWithinLimits : BOOL;
  checkTargetStateWithinLimits : BOOL;
END_VAR
VAR
  stateMem : TrajectoryState;
END_VAR
stateMem := _state;
ValidateInput := ValidateInputOrAbort(checkCurrentStateWithinLimits, checkTargetStateWithinLimits);
_state := stateMem;
END_METHOD

/// \copydoc Struckig.Otg#ValidateInput
{attribute 'conditionalshow'}
METHOD PROTECTED ValidateInputOrAbort : BOOL
VAR_INPUT
  checkCurrentStateWithinLimits : BOOL;
  checkTargetStateWithinLimits : BOOL;
END_VAR
VAR
  i, dofsEnd : INT;
  aMin, vMin, a0, af, v0, vf : LREAL;
  ci : ControlInterfaceType;
END_VAR
IF Dofs = 0
THEN
  RETURN;
END_IF

dofsEnd := Dofs-1;
FOR i:=0 TO dofsEnd
DO

  IF MaxJerk[i] <> MaxJerk[i] OR_ELSE // isnan
     MaxJerk[i] < 0.0
  THEN
    AbortErrorId(TrajectoryErrorCode.InvalidInput, 'maximum jerk limit should be larger than or equal to zero');
    RETURN;
	END_IF

  IF MaxAcceleration[i] <> MaxAcceleration[i] OR_ELSE // isnan
     MaxAcceleration[i] < 0.0
  THEN
    AbortErrorId(TrajectoryErrorCode.InvalidInput, 'maximum acceleration limit should be larger than or equal to zero'); 
    RETURN;
  END_IF

  aMin := SEL(MinAcceleration[i] = 0, MinAcceleration[i] ,-MaxAcceleration[i]);
  IF aMin <> aMin OR_ELSE // isnan  
     aMin > 0
  THEN    
    AbortErrorId(TrajectoryErrorCode.InvalidInput, 'minimum acceleration limit should be smaller than or equal zero'); 
    RETURN;
  END_IF
  
  a0 := CurrentAcceleration[i];
  IF a0 <> a0 // isnan
  THEN
    AbortErrorId(TrajectoryErrorCode.InvalidInput, 'current acceleration should be a valid number'); 
    RETURN;
	END_IF
  
  af := TargetAcceleration[i];
  IF af <> af // isnan
  THEN
    AbortErrorId(TrajectoryErrorCode.InvalidInput, 'target acceleration should be a valid number'); 
    RETURN;
	END_IF  
  
  IF checkCurrentStateWithinLimits
  THEN
    IF a0 > MaxAcceleration[i]
    THEN
      AbortErrorId(TrajectoryErrorCode.InvalidInput, 'current acceleration exceeds its maximum acceleration limit'); 
      RETURN;
    END_IF
    
    IF  a0 < aMin
    THEN 
      AbortErrorId(TrajectoryErrorCode.InvalidInput, 'current acceleration undercuts its minimum acceleration limit'); 
      RETURN;
    END_IF    
  END_IF
  
  IF checkTargetStateWithinLimits 
  THEN
    IF af > MaxAcceleration[i]
    THEN
      AbortErrorId(TrajectoryErrorCode.InvalidInput, 'target acceleration exceeds its maximum acceleration limit'); 
      RETURN;
    END_IF
 
    IF af < aMin
    THEN
      AbortErrorId(TrajectoryErrorCode.InvalidInput, 'target acceleration undercuts its minimum acceleration limit'); 
      RETURN;  
		END_IF
  END_IF
  
  v0 := CurrentVelocity[i];
  IF v0 <> v0// isnan
  THEN
    AbortErrorId(TrajectoryErrorCode.InvalidInput, 'current velocity should be a valid number'); 
    RETURN;
	END_IF
  
  vf := TargetVelocity[i];
  IF vf <> vf // isnan
  THEN
    AbortErrorId(TrajectoryErrorCode.InvalidInput, 'target velocity should be a valid number'); 
    RETURN;
	END_IF
  
  ci := SEL(PerDofControlInterface[i] = ControlInterfaceType.Undefined, PerDofControlInterface[i], ControlInterface);
  IF (ci = ControlInterfaceType.Position)
  THEN
  
    IF CurrentPosition[i] <> CurrentPosition[i] //isnan
    THEN
      AbortErrorId(TrajectoryErrorCode.InvalidInput, 'current position should be a valid number'); 
      RETURN;
    END_IF
    
    IF TargetPosition[i] <> TargetPosition[i] //isnan
    THEN
      AbortErrorId(TrajectoryErrorCode.InvalidInput, 'target position should be a valid number'); 
      RETURN;
    END_IF    
    
    IF MaxVelocity[i] <> MaxVelocity[i] OR_ELSE // isnan
       MaxVelocity[i] < 0.0      
    THEN
      AbortErrorId(TrajectoryErrorCode.InvalidInput, 'maximum velocity limit should be larger than or equal to zero'); 
      RETURN;
		END_IF
    
    vMin := SEL(MinVelocity[i] = 0, MinVelocity[i], -MaxVelocity[i]);
    IF vMin <> vMin OR_ELSE // isnan
       vMin > 0.0
    THEN
      AbortErrorId(TrajectoryErrorCode.InvalidInput, 'minimum velocity limit should be smaller than or equal to zero'); 
      RETURN;
    END_IF
    
    IF checkCurrentStateWithinLimits 
    THEN
      IF v0 > MaxVelocity[i]
      THEN
        AbortErrorId(TrajectoryErrorCode.InvalidInput, 'current velocity exceeds its maximum velocity limit'); 
        RETURN;
      END_IF

      IF v0 < vMin
      THEN
        AbortErrorId(TrajectoryErrorCode.InvalidInput, 'current velocity undercuts its minimum velocity limit'); 
        RETURN;
      END_IF
    END_IF
    
    IF checkTargetStateWithinLimits
    THEN
      IF vf > MaxVelocity[i]
      THEN
        AbortErrorId(TrajectoryErrorCode.InvalidInput, 'target velocity exceeds its maximum velocity limit'); 
        RETURN;
      END_IF
      
      IF vf < vMin
      THEN
        AbortErrorId(TrajectoryErrorCode.InvalidInput, 'target velocity undercuts its minimum velocity limit'); 
        RETURN;
			END_IF
    END_IF
    
    IF checkCurrentStateWithinLimits
    THEN
      IF a0 > 0 AND_THEN MaxJerk[i] > 0 AND_THEN VelocityAtZero(v0, a0, MaxJerk[i]) > MaxVelocity[i]
      THEN
        AbortErrorId(TrajectoryErrorCode.InvalidInput, 'Trajectory will inevitably reach a velocity from the current kinematic state that will exceed its maximum velocity limit'); 
        RETURN;
			END_IF
      
      IF a0 < 0 AND_THEN MaxJerk[i] > 0 AND_THEN VelocityAtZero(v0, a0, -MaxJerk[i]) < vMin
      THEN
        AbortErrorId(TrajectoryErrorCode.InvalidInput, 'Trajectory will inevitably reach a velocity from the current kinematic state that will undercut its minimum velocity limit'); 
        RETURN;
			END_IF      
    END_IF
    
    IF checkTargetStateWithinLimits
    THEN
      IF af < 0 AND_THEN MaxJerk[i] > 0 AND_THEN VelocityAtZero(vf, af, MaxJerk[i]) > MaxVelocity[i]
      THEN
        AbortErrorId(TrajectoryErrorCode.InvalidInput, 'Trajectory will inevitably reach a velocity from the current kinematic state that will exceed its maximum velocity limit'); 
        RETURN;
			END_IF
      
      IF af > 0 AND_THEN MaxJerk[i] > 0 AND_THEN VelocityAtZero(vf, af, -MaxJerk[i]) < vMin
      THEN
        AbortErrorId(TrajectoryErrorCode.InvalidInput, 'Trajectory will inevitably reach a velocity from the current kinematic state that will undercut its minimum velocity limit'); 
        RETURN;
			END_IF  
    END_IF    
  END_IF

END_FOR

IF CycleTime <= 0 AND_THEN Discretization <> DiscretizationType.Continuous
THEN
  AbortErrorId(TrajectoryErrorCode.InvalidInput, 'Cycle time parameter should be larger than zero'); 
  RETURN;
END_IF

ValidateInputOrAbort := TRUE;
END_METHOD

METHOD INTERNAL VelocityAtZero : LREAL
VAR_INPUT
  v0 : LREAL;
  a0 : LREAL;
  j : LREAL;
END_VAR
VelocityAtZero := v0 + (a0 * a0)/(2 * j);
END_METHOD

END_FUNCTION_BLOCK
